{attribute addProperty BoxType "AT2050-0501-0021"}
{attribute addProperty Id "A_0086_AT2050_5500_0019_AT2050_5500AT2050_3DCFC8D064080"}
{attribute addProperty CRC "3240237556"}
{attribute addProperty SizeInBites "640"}
{attribute addProperty SizeInBytes "80"}
TYPE A_0058_AT2050_0501_0021_C12219F4 EXTENDS AT2050_9506A482 :
STRUCT
	{attribute addProperty Name "A_0086_AT2050_5500_0019_AT2050_5500"}
	A_0086_AT2050_5500_0019_AT2050_5500 : AT2050_3DCFC8D0;
END_STRUCT
END_TYPE

(* stored: Version 1.2.0.0, ProductVersion 3.1.4024.9
   DUT A_0058_AT2050_0501_0021_C12219F4: Id {4d58cc30-c190-4d42-a3dc-caaa2b4126a8} *)
